// TIA Portal V17 export
// export: Created 2024-08-07T21:44:08.5065949Z, ExportSetting WithDefaults, DisplayName Totally Integrated Automation Portal, DisplayVersion V17 Update 7, DisplayName TIA Portal Openness, DisplayVersion V17 Update 7, DisplayName TIA Portal Version Control Interface, DisplayVersion V17, DisplayName SINAMICS Startdrive Advanced, DisplayVersion V17 SP2, DisplayName SINAMICS Startdrive G110M, G120, G120C, G120D, G120P, G115D, DisplayVersion V17 SP2, DisplayName SINAMICS Startdrive G130, G150, S120, S150, SINAMICS MV, S210, DisplayVersion V17 SP2, DisplayName STEP 7 Professional, DisplayVersion V17 Update 7, DisplayName STEP 7 Safety, DisplayVersion V17 Update 6, DisplayName WinCC Advanced / Unified PC, DisplayVersion V17 Update 7
DATA_BLOCK "Main_Safety_RTG1_DB"   // DB48, F_DB
NAME : FUSI
VERSION : 0.1
// stored: AutoNumber true, DBAccessibleFromOPCUA true, DBAccessibleFromWebserver true, InstanceOfName Main_Safety_RTG1, InstanceOfType FB
"Main_Safety_RTG1"
   // VAR
   //    ACK_GL_Instance : ACK_GL;
   //    "ESTOP1_3L+" : ESTOP1;
   //    "FDBACK_A2.7" : FDBACK;
   //    "ESTOP1_4L+" : ESTOP1;
   //    "FDBACK_A2.8" : FDBACK;
   //    "FDBACK_A2.9" : FDBACK;
   //    "ESTOP1_5L+" : ESTOP1;
   //    "F_IEC_Timer_3L+" : TON;
   //    "F_IEC_Timer_4L+" : TON;
   //    FDBACK_KF101x : FDBACK;
   //    FDBACK_KM20_KM21 : FDBACK;
   // END_VAR
BEGIN
END_DATA_BLOCK
